ABB RAPID module: ReplayTargets_v14.mod

MODULE ReplayTargets_v14
    ! Generated from tests_v14.csv and success_v14.csv.
    ! Target names include version and testId. B* variants include version, testId, and confId.

    ! Robtargets and jointtargets for replay
    CONST robtarget rA_v14_t1 := [[1867.5,0,1823],[2.18557E-8,0,-1,0],[0,0,0,0],[9E+09,9E+09,9E+09,9E+09,9E+09,9E+09]];
    CONST robtarget rB_v14_t1 := [[1496.97,1618.25,1827.16],[0.0677417,0.105668,0.725414,0.676771],[0,-3,-5,0],[9E+09,9E+09,9E+09,9E+09,9E+09,9E+09]];
    CONST robtarget rB_v14_t1_c4 := [[1496.97,1618.25,1827.16],[0.0677417,0.105668,0.725414,0.676771],[0,-4,0,0],[9E+09,9E+09,9E+09,9E+09,9E+09,9E+09]];
    CONST robtarget rB_v14_t1_c5 := [[1496.97,1618.25,1827.16],[0.0677417,0.105668,0.725414,0.676771],[0,0,0,0],[9E+09,9E+09,9E+09,9E+09,9E+09,9E+09]];
    CONST jointtarget jA_v14_t1 := [[0,-2.3802E-6,7.25062E-7,0,90,0],[9E+09,9E+09,9E+09,9E+09,9E+09,9E+09]];
    CONST jointtarget jB_v14_t1 := [[44.9999,9.3,-4.3,-270,30.9,-360.001],[9E+09,9E+09,9E+09,9E+09,9E+09,9E+09]];
    CONST jointtarget jBseed_v14_t1 := [[45,9.3,-4.3,-270,30.9,-360],[9E+09,9E+09,9E+09,9E+09,9E+09,9E+09]];
    CONST num seedB_v14_t1 := 23768;

    CONST robtarget rA_v14_t5 := [[-101.745,-532.207,3241.29],[0.68387,0.621186,-0.113478,-0.365475],[-1,-1,0,0],[9E+09,9E+09,9E+09,9E+09,9E+09,9E+09]];
    CONST robtarget rB_v14_t5 := [[1262.13,1262.13,-115.711],[0.183484,0.335827,0.810765,0.44296],[0,-2,-2,0],[9E+09,9E+09,9E+09,9E+09,9E+09,9E+09]];
    CONST robtarget rB_v14_t5_c7 := [[1262.13,1262.13,-115.711],[0.183484,0.335827,0.810765,0.44296],[0,-4,4,0],[9E+09,9E+09,9E+09,9E+09,9E+09,9E+09]];
    CONST jointtarget jA_v14_t5 := [[-89.9997,-20.3,-44.7,-45.0005,59.5,89.9995],[9E+09,9E+09,9E+09,9E+09,9E+09,9E+09]];
    CONST jointtarget jB_v14_t5 := [[45,46.1,31.9,-180,45.3,-90.0007],[9E+09,9E+09,9E+09,9E+09,9E+09,9E+09]];
    CONST jointtarget jBseed_v14_t5 := [[45,46.1,31.9,-180,45.3,-90],[9E+09,9E+09,9E+09,9E+09,9E+09,9E+09]];
    CONST num seedB_v14_t5 := 11381;

    CONST robtarget rA_v14_t6 := [[1262.13,1262.13,-115.711],[0.183484,0.335827,0.810765,0.44296],[0,-2,-2,0],[9E+09,9E+09,9E+09,9E+09,9E+09,9E+09]];
    CONST robtarget rB_v14_t6 := [[50.466,1991.61,1060.33],[0.133544,0.0746247,0.862646,0.482119],[1,-2,-2,0],[9E+09,9E+09,9E+09,9E+09,9E+09,9E+09]];
    CONST robtarget rB_v14_t6_c2 := [[50.466,1991.61,1060.33],[0.133544,0.0746247,0.862646,0.482119],[0,0,-4,0],[9E+09,9E+09,9E+09,9E+09,9E+09,9E+09]];
    CONST robtarget rB_v14_t6_c3 := [[50.466,1991.61,1060.33],[0.133544,0.0746247,0.862646,0.482119],[0,4,-4,0],[9E+09,9E+09,9E+09,9E+09,9E+09,9E+09]];
    CONST jointtarget jA_v14_t6 := [[45,46.1,31.9,-180,45.3,-90.0007],[9E+09,9E+09,9E+09,9E+09,9E+09,9E+09]];
    CONST jointtarget jB_v14_t6 := [[90.0009,5.8,25.8,-90.0009,17.6,-180],[9E+09,9E+09,9E+09,9E+09,9E+09,9E+09]];
    CONST jointtarget jBseed_v14_t6 := [[90,5.8,25.8,-90,17.6,-180],[9E+09,9E+09,9E+09,9E+09,9E+09,9E+09]];
    CONST num seedB_v14_t6 := 8398;

    CONST robtarget rA_v14_t10 := [[-1385.59,1483.98,2775.73],[0.736409,-0.295405,0.188582,0.578683],[1,-2,1,0],[9E+09,9E+09,9E+09,9E+09,9E+09,9E+09]];
    CONST robtarget rB_v14_t10 := [[96.7425,1721.93,2800.28],[0.921685,-0.0636439,0.327855,0.197374],[0,-2,-4,0],[9E+09,9E+09,9E+09,9E+09,9E+09,9E+09]];
    CONST robtarget rB_v14_t10_c5 := [[96.7425,1721.93,2800.28],[0.921685,-0.0636439,0.327855,0.197374],[0,0,0,0],[9E+09,9E+09,9E+09,9E+09,9E+09,9E+09]];
    CONST jointtarget jA_v14_t10 := [[135,19,-47.8,-135,36.1,90.0002],[9E+09,9E+09,9E+09,9E+09,9E+09,9E+09]];
    CONST jointtarget jB_v14_t10 := [[89.9996,3.8,-30.9,-134.999,55,-270.001],[9E+09,9E+09,9E+09,9E+09,9E+09,9E+09]];
    CONST jointtarget jBseed_v14_t10 := [[90,3.8,-30.9,-135,55,-270],[9E+09,9E+09,9E+09,9E+09,9E+09,9E+09]];
    CONST num seedB_v14_t10 := 1010;

    CONST robtarget rA_v14_t11 := [[96.7425,1721.93,2800.28],[0.921685,-0.0636439,0.327855,0.197374],[0,-2,-4,0],[9E+09,9E+09,9E+09,9E+09,9E+09,9E+09]];
    CONST robtarget rB_v14_t11 := [[89.2692,188.834,2998.51],[0.973387,-0.190673,-0.110388,0.0630517],[0,-3,2,0],[9E+09,9E+09,9E+09,9E+09,9E+09,9E+09]];
    CONST robtarget rB_v14_t11_c1 := [[89.2692,188.834,2998.51],[0.973387,-0.190673,-0.110388,0.0630517],[0,-4,-4,0],[9E+09,9E+09,9E+09,9E+09,9E+09,9E+09]];
    CONST robtarget rB_v14_t11_c2 := [[89.2692,188.834,2998.51],[0.973387,-0.190673,-0.110388,0.0630517],[0,0,-4,0],[9E+09,9E+09,9E+09,9E+09,9E+09,9E+09]];
    CONST jointtarget jA_v14_t11 := [[89.9996,3.8,-30.9,-134.999,55,-270.001],[9E+09,9E+09,9E+09,9E+09,9E+09,9E+09]];
    CONST jointtarget jB_v14_t11 := [[44.9991,-46.5,-10.5,-225,36.6,180],[9E+09,9E+09,9E+09,9E+09,9E+09,9E+09]];
    CONST jointtarget jBseed_v14_t11 := [[45,-46.5,-10.5,-225,36.6,180],[9E+09,9E+09,9E+09,9E+09,9E+09,9E+09]];
    CONST num seedB_v14_t11 := 31540;

    CONST robtarget rA_v14_t13 := [[-1547.23,-1520.12,2800.65],[0.364982,-0.219726,-0.396204,0.813346],[-2,-2,-4,0],[9E+09,9E+09,9E+09,9E+09,9E+09,9E+09]];
    CONST robtarget rB_v14_t13 := [[0.00721235,-1337.1,3323.94],[0.381423,0.031026,-0.0748968,0.920839],[-1,1,0,0],[9E+09,9E+09,9E+09,9E+09,9E+09,9E+09]];
    CONST robtarget rB_v14_t13_c1 := [[0.00721235,-1337.1,3323.94],[0.381423,0.031026,-0.0748968,0.920839],[0,-4,-4,0],[9E+09,9E+09,9E+09,9E+09,9E+09,9E+09]];
    CONST jointtarget jA_v14_t13 := [[-134.999,31.7,-68.1,-90,6.6,-360],[9E+09,9E+09,9E+09,9E+09,9E+09,9E+09]];
    CONST jointtarget jB_v14_t13 := [[-89.9997,19.4,-78.7,179.999,21.4,45.0005],[9E+09,9E+09,9E+09,9E+09,9E+09,9E+09]];
    CONST jointtarget jBseed_v14_t13 := [[-90,19.4,-78.7,180,21.4,45],[9E+09,9E+09,9E+09,9E+09,9E+09,9E+09]];
    CONST num seedB_v14_t13 := 27689;

ENDMODULE
